FUNCTION_BLOCK FB_BufferA_TestControl
VAR_INPUT
    BufferA   : ITF_BufferA;        // equipment
    TestState : E_PackMLStates;      // welke state wil je sturen
END_VAR
VAR
    _LastCmd  : E_PackMLStates := E_PackMLStates.Idle;
END_VAR

// Stuur alleen een nieuwe command-state als TestState verandert
IF TestState <> _LastCmd THEN
    BufferA.InputState := TestState;
    _LastCmd := TestState;
END_IF;

END_FUNCTION_BLOCK

(* stored: Version 1.1.0.1
   POU FB_BufferA_TestControl: Id {a408d9d4-03ff-442e-b9d9-79c94b6d179a}, SpecialFunc None *)
